// Block: Area04_Messages

DATA_BLOCK Area04_Messages
VERSION : 0.1
   NON_RETAIN
   VAR
      A : Struct
         Msg : Array[1..400] of Bool;
         Hmi : Array[1..25] of Word;
         Ack : Array[1..25] of Word;
      END_STRUCT;
      W : Struct
         Msg : Array[1..400] of Bool;
         Hmi : Array[1..25] of Word;
         Ack : Array[1..25] of Word;
      END_STRUCT;
   END_VAR

BEGIN
   // No initialization required
END_DATA_BLOCK
